INTERFACE I_CyclicCall

METHOD CyclicCall
END_METHOD

END_INTERFACE

(* stored: Version 1.1.0.1, ProductVersion 3.1.4024.11
   Itf I_CyclicCall: Id {98176e96-c0c9-4724-813d-30bdf1a5be00}
   Method CyclicCall: Id {61ffef0b-4a25-445e-a86a-76c2c3276504} *)
